{attribute 'qualified_only'}
VAR_GLOBAL RETAIN
	Actual_GLV_State :INT:=-1;
	Actual_In_State: INT:=-1;

END_VAR

(* stored: Version 1.1.0.1, ProductVersion 3.1.4024.4
   GVL UR3RetVarState: Id {4339c6cc-5443-4b9b-ab6e-006fb0eea905} *)
